FUNCTION F_ITC_SendRAQ : BOOL
(**************************************************************************************
 * 	Application		:	BoxControl Framework
 *	Revision		:	$Revision: 404529 $
 *	Revision date	:	$Date: 2018-04-23 08:21:38 +0200 (Mo., 23 Apr 2018) $
 *	Last changed by	:	$Author: b7bolm $
 *	URL				:	$URL: http://almscdc.swisslog.com/repo/SWPD/Development/BoxControlFramework/20_Release/trunk/01_Software/BCF/BCF/JumpStart/20_Product/10_App/11_Com/10_Lib/10_Conv/11_ITC/F_ITC_SendRAQ.TcPOU $
 *
 *	Purpose			:	Wrap message - RAQ
 *
 * ------------------------------------------------------------------------------------
 *	Copyright Swisslog [IP AG], Switzerland. All rights reserved.
 * 
 * ------------------------------------------------------------------------------------
 *	
 * 	Revision History: 
 *
 * 	VERSION			DATE			INITIALS			DESCRIPTION
 *	0.1				01.01.2001		swl					Example
 *
 **************************************************************************************)
VAR_INPUT
	eChannelSrc				: E_MFCS_Channel; // Source communicaton channel
	PositionName			: STRING(Conveyor.POSITION_STRINGLENGTH); // SIS MM-GGG-EEEE-FF-Z
	GroupID					: ULINT;
	NumberOfRA				: INT;
END_VAR
VAR
	RAQ						: ST_ITC_RAQ; 
END_VAR

// Map values
RAQ.Position := PositionName;
RAQ.GroupID := GroupID;
RAQ.NumberOfRA := NumberOfRA;

// Forward to ITC
F_ITC_SendRAQ := fbITC_Manager.M_SendData(
					meChannel	:= eChannelSrc,
					mMsgType	:= E_ITC_MsgTypeConv.ROBOT_ACTION_REQUEST,
					mpData		:= ADR(RAQ),
					mLen		:= SIZEOF(RAQ));

END_FUNCTION

(* stored: Version 1.1.0.1, ProductVersion 3.1.4022.12
   POU F_ITC_SendRAQ: Id {34ff58e1-b80e-4e4d-bd39-3595b728d625}, SpecialFunc None *)
